FUNCTION_BLOCK FB_OutLinear
VAR
	//Properties
	bError 				: BOOL 				:= FALSE;
	stIOConv			: IO_TERMINAL_PARAMETERS;
	
	//value
	fValueOut			: REAL;
	
	//Raw value
	nValueOutRaw		AT %Q* : INT;
END_VAR

PROPERTY Error : BOOL
GET
Error := THIS^.bError;
END_GET
SET
THIS^.bError := Error;
END_SET
END_PROPERTY

PROPERTY IO_Conversion : REFERENCE TO IO_TERMINAL_PARAMETERS
GET
IO_Conversion REF= THIS^.stIOConv;
END_GET
SET
THIS^.stIOConv := IO_Conversion;
END_SET
END_PROPERTY

PROPERTY ValueOut : REAL
GET
ValueOut := THIS^.fValueOut;
END_GET
SET
THIS^.fValueOut := ValueOut;
END_SET
END_PROPERTY

METHOD Write
nValueOutRaw := REAL_TO_INT(F_LIN2(X:=fValueOut,X1:=stIOConv.cValue1,Y1:=stIOConv.cValue1Raw,X2:=stIOConv.cValue2,Y2:=stIOConv.cValue2Raw));
END_METHOD

END_FUNCTION_BLOCK

(* stored: Version 1.1.0.1, ProductVersion 3.1.4024.3
   POU FB_OutLinear: Id {1129039b-235d-42f6-9031-f7cf02c75c4f}, SpecialFunc None
   Property Error: Id {c75753be-259e-41d7-a0dd-7398f9503b9a}
   Get Get: Id {12324abb-39dd-4ba1-96d6-af83bbf38b7e}
   Set Set: Id {a3dfe7d4-d0a0-48fa-b801-050d29862b03}
   Property IO_Conversion: Id {95b1d063-2aea-4a38-a4a7-324d5c8b277a}
   Get Get: Id {47991903-5933-4c6e-91e5-796a5cc199c1}
   Set Set: Id {134f0b25-5d4e-4b08-bab8-149e7c7408dc}
   Property ValueOut: Id {98ce44bc-1da4-4c29-ba1b-87cfea33daef}
   Get Get: Id {625a6961-46ca-4f32-85e4-555bebedf209}
   Set Set: Id {536de769-5b2d-4c40-a418-3ced6a3f8fc9}
   Method Write: Id {4ea49992-efbe-4dbe-abec-201d6b60ac5f} *)
